// TIA Portal V20 export
VAR_GLOBAL   // PLC tag table "Table de variables_1"
   "E0.0" AT %I0.0 : Bool;
   "E0.1" AT %I0.1 : Bool;
   "E0.2" AT %I0.2 : Bool;
   "E0.3" AT %I0.3 : Bool;
   "M2.0" AT %I0.4 : Bool;
   "M2.1" AT %I0.5 : Bool;
END_VAR
